DATA_BLOCK "IO"
TITLE = A-io
{ S7_Optimized_Access := 'TRUE' }
AUTHOR : PiotrSlezak
FAMILY : Vorster
VERSION : 0.1
   STRUCT
      io { S7_SetPoint := 'False'} : Array[0..17] of "Tio";
	  alarm { S7_SetPoint := 'True'} : Array[0..2] of UInt;
   END_STRUCT;


BEGIN

END_DATA_BLOCK

